{attribute 'GeneratedUsingTerminal: KL1184'}
{attribute addProperty BoxType "KL1184"}
{attribute addProperty Id "Channel_1AT %I*Channel_87C95E760Channel_2AT %I*Channel_87C95E760Channel_3AT %I*Channel_87C95E760Channel_4AT %I*Channel_87C95E760"}
{attribute addProperty CRC "1243970859"}
{attribute addProperty Size "0"}
TYPE KL1184_4A257D2B :
STRUCT
	{attribute addProperty Name "Channel_1"}
	Channel_1 : Channel_87C95E76;
	{attribute addProperty Name "Channel_2"}
	Channel_2 : Channel_87C95E76;
	{attribute addProperty Name "Channel_3"}
	Channel_3 : Channel_87C95E76;
	{attribute addProperty Name "Channel_4"}
	Channel_4 : Channel_87C95E76;
END_STRUCT
END_TYPE

(* stored: Version 1.2.0.0, ProductVersion 3.1.4024.9
   DUT KL1184_4A257D2B: Id {88504116-8830-406e-9f0a-c1ef37e01689} *)
